# EPICS StreamDevice protocol: streamDevice/alex.proto
# Alex's Sidekick EPICS protocol file
# Built by examining examples at: https://paulscherrerinstitute.github.io/StreamDevice/protocol.html#gen

Terminator = LF;

info {
	ExtraInput = Ignore;
	out "*IDN?";
	in "%39c";
}

setCycle {
	ExtraInput = Ignore;
	out "POS:CYC %u";
}

debug {
   ExtraInput = Ignore;
   out "%s";
   in "%39c";
}
